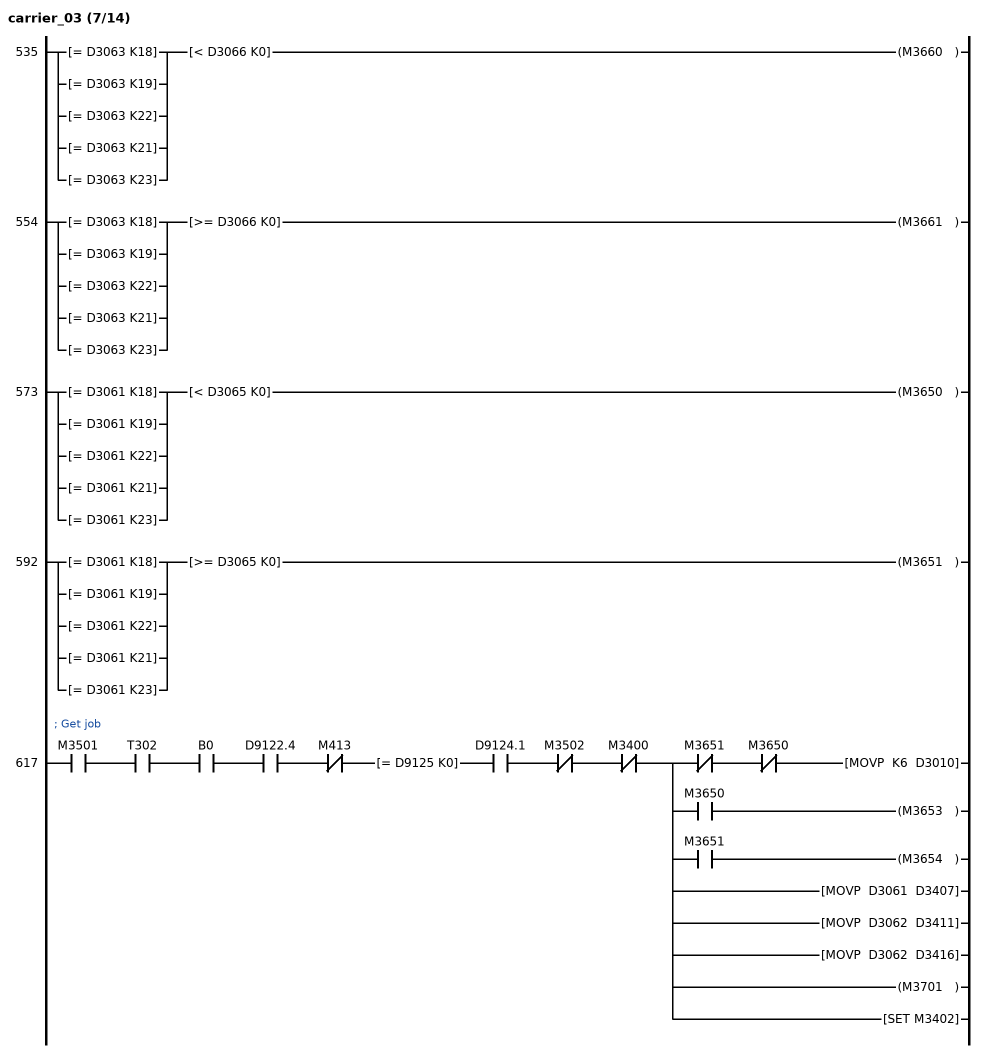
[picture p72: ladder of carrier_03, rungs at steps 535 to 617]
535   LD=     D3063 K18
      OR=     D3063 K19
      OR=     D3063 K22
      OR=     D3063 K21
      OR=     D3063 K23
      AND<    D3066 K0
      OUT     M3660
554   LD=     D3063 K18
      OR=     D3063 K19
      OR=     D3063 K22
      OR=     D3063 K21
      OR=     D3063 K23
      AND>=   D3066 K0
      OUT     M3661
573   LD=     D3061 K18
      OR=     D3061 K19
      OR=     D3061 K22
      OR=     D3061 K21
      OR=     D3061 K23
      AND<    D3065 K0
      OUT     M3650
592   LD=     D3061 K18
      OR=     D3061 K19
      OR=     D3061 K22
      OR=     D3061 K21
      OR=     D3061 K23
      AND>=   D3065 K0
      OUT     M3651
; Get job
617   LD      M3501
      AND     T302
      AND     B0
      AND     D9122.4
      ANI     M413
      AND=    D9125 K0
      AND     D9124.1
      ANI     M3502
      ANI     M3400
      MPS
      ANI     M3651
      ANI     M3650
      MOVP    K6 D3010
      MRD
      AND     M3650
      OUT     M3653
      MRD
      AND     M3651
      OUT     M3654
      MPP
      MOVP    D3061 D3407
      MOVP    D3062 D3411
      MOVP    D3062 D3416
      OUT     M3701
      SET     M3402
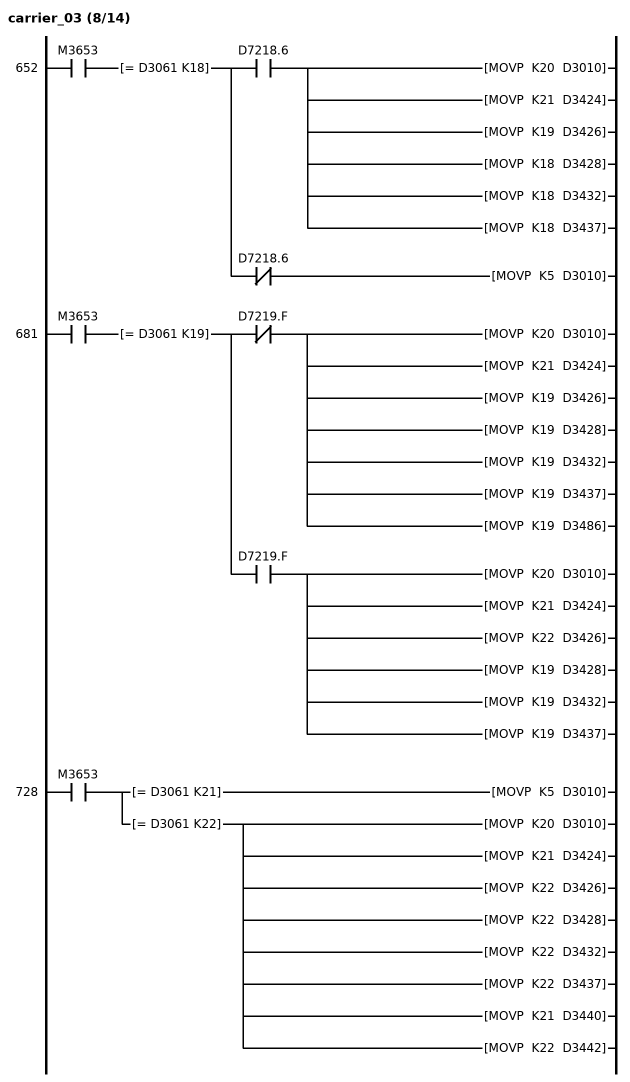
652   LD      M3653
      AND=    D3061 K18
      MPS
      AND     D7218.6
      MOVP    K20 D3010
      MOVP    K21 D3424
      MOVP    K19 D3426
      MOVP    K18 D3428
      MOVP    K18 D3432
      MOVP    K18 D3437
      MPP
      ANI     D7218.6
      MOVP    K5 D3010
681   LD      M3653
      AND=    D3061 K19
      MPS
      ANI     D7219.F
      MOVP    K20 D3010
      MOVP    K21 D3424
      MOVP    K19 D3426
      MOVP    K19 D3428
      MOVP    K19 D3432
      MOVP    K19 D3437
      MOVP    K19 D3486
      MPP
      AND     D7219.F
      MOVP    K20 D3010
      MOVP    K21 D3424
      MOVP    K22 D3426
      MOVP    K19 D3428
      MOVP    K19 D3432
      MOVP    K19 D3437
728   LD      M3653
      MPS
      AND=    D3061 K21
      MOVP    K5 D3010
      MPP
      AND=    D3061 K22
      MOVP    K20 D3010
      MOVP    K21 D3424
      MOVP    K22 D3426
      MOVP    K22 D3428
      MOVP    K22 D3432
      MOVP    K22 D3437
      MOVP    K21 D3440
      MOVP    K22 D3442
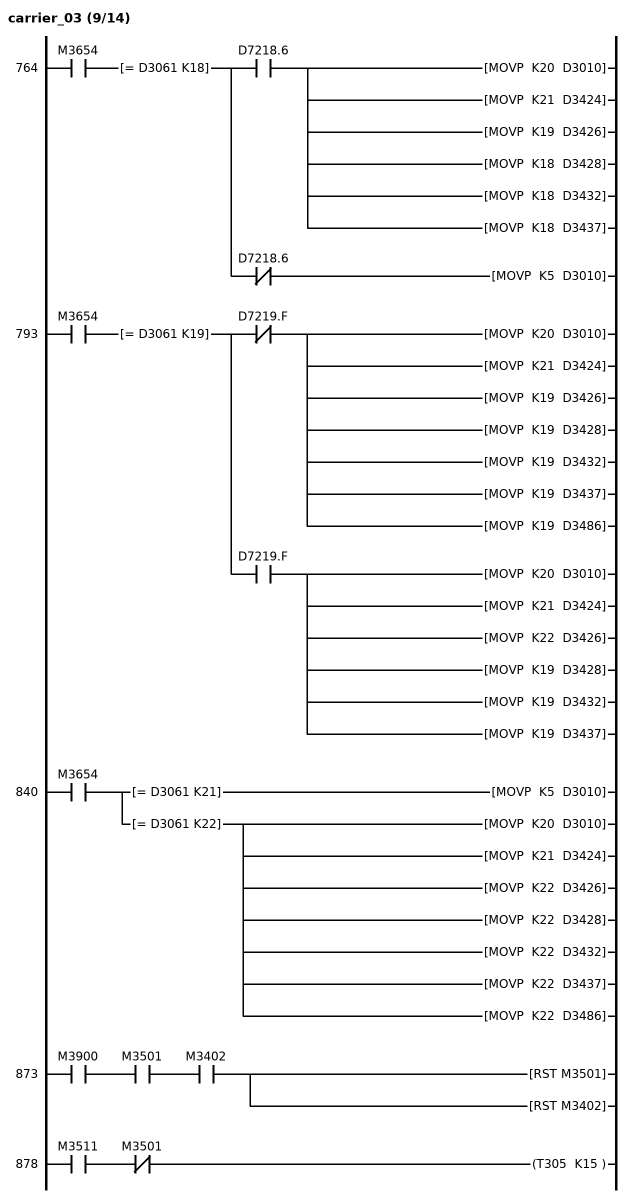
764   LD      M3654
      AND=    D3061 K18
      MPS
      AND     D7218.6
      MOVP    K20 D3010
      MOVP    K21 D3424
      MOVP    K19 D3426
      MOVP    K18 D3428
      MOVP    K18 D3432
      MOVP    K18 D3437
      MPP
      ANI     D7218.6
      MOVP    K5 D3010
793   LD      M3654
      AND=    D3061 K19
      MPS
      ANI     D7219.F
      MOVP    K20 D3010
      MOVP    K21 D3424
      MOVP    K19 D3426
      MOVP    K19 D3428
      MOVP    K19 D3432
      MOVP    K19 D3437
      MOVP    K19 D3486
      MPP
      AND     D7219.F
      MOVP    K20 D3010
      MOVP    K21 D3424
      MOVP    K22 D3426
      MOVP    K19 D3428
      MOVP    K19 D3432
      MOVP    K19 D3437
840   LD      M3654
      MPS
      AND=    D3061 K21
      MOVP    K5 D3010
      MPP
      AND=    D3061 K22
      MOVP    K20 D3010
      MOVP    K21 D3424
      MOVP    K22 D3426
      MOVP    K22 D3428
      MOVP    K22 D3432
      MOVP    K22 D3437
      MOVP    K22 D3486
873   LD      M3900
      AND     M3501
      AND     M3402
      RST     M3501
      RST     M3402
878   LD      M3511
      ANI     M3501
      OUT     T305 K15
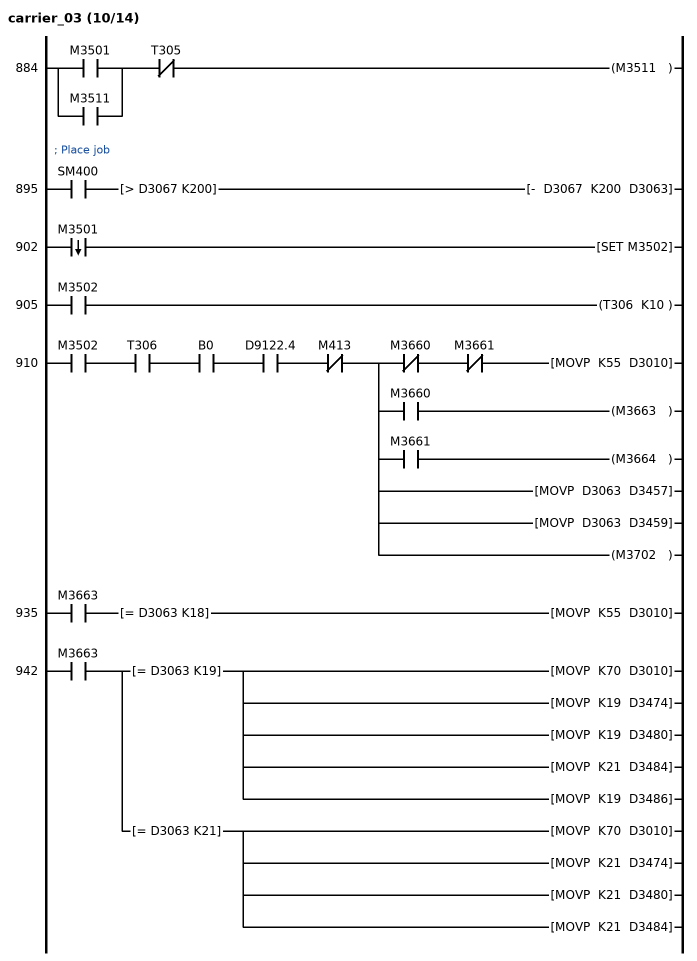
884   LD      M3501
      OR      M3511
      ANI     T305
      OUT     M3511
; Place job
895   LD      SM400
      AND>    D3067 K200
      -       D3067 K200 D3063
902   LDF     M3501
      SET     M3502
905   LD      M3502
      OUT     T306 K10
910   LD      M3502
      AND     T306
      AND     B0
      AND     D9122.4
      ANI     M413
      MPS
      ANI     M3660
      ANI     M3661
      MOVP    K55 D3010
      MRD
      AND     M3660
      OUT     M3663
      MRD
      AND     M3661
      OUT     M3664
      MPP
      MOVP    D3063 D3457
      MOVP    D3063 D3459
      OUT     M3702
935   LD      M3663
      AND=    D3063 K18
      MOVP    K55 D3010
942   LD      M3663
      MPS
      AND=    D3063 K19
      MOVP    K70 D3010
      MOVP    K19 D3474
      MOVP    K19 D3480
      MOVP    K21 D3484
      MOVP    K19 D3486
      MPP
      AND=    D3063 K21
      MOVP    K70 D3010
      MOVP    K21 D3474
      MOVP    K21 D3480
      MOVP    K21 D3484
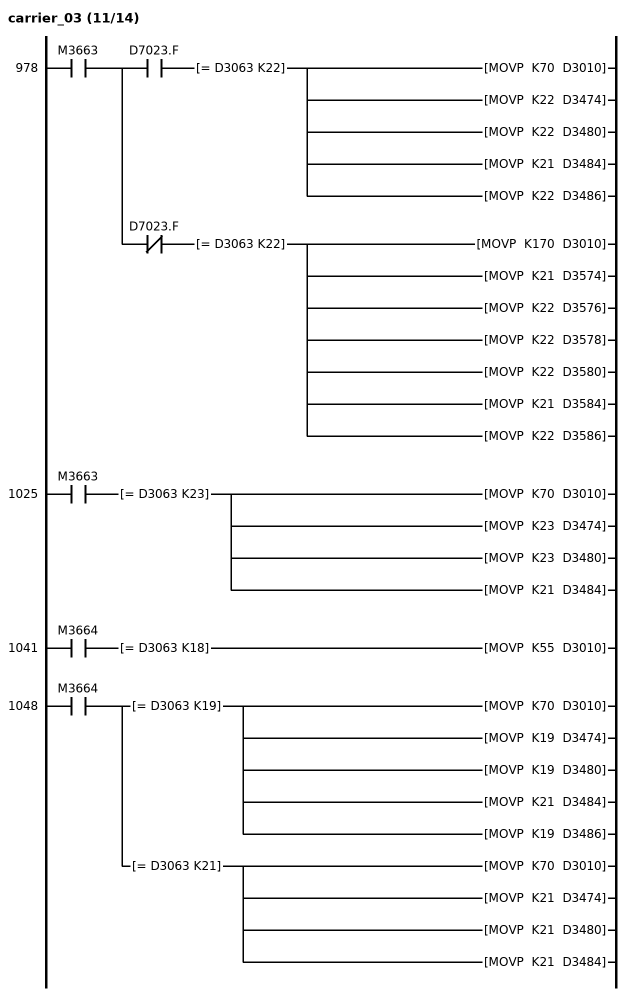
978   LD      M3663
      MPS
      AND     D7023.F
      AND=    D3063 K22
      MOVP    K70 D3010
      MOVP    K22 D3474
      MOVP    K22 D3480
      MOVP    K21 D3484
      MOVP    K22 D3486
      MPP
      ANI     D7023.F
      AND=    D3063 K22
      MOVP    K170 D3010
      MOVP    K21 D3574
      MOVP    K22 D3576
      MOVP    K22 D3578
      MOVP    K22 D3580
      MOVP    K21 D3584
      MOVP    K22 D3586
1025  LD      M3663
      AND=    D3063 K23
      MOVP    K70 D3010
      MOVP    K23 D3474
      MOVP    K23 D3480
      MOVP    K21 D3484
1041  LD      M3664
      AND=    D3063 K18
      MOVP    K55 D3010
1048  LD      M3664
      MPS
      AND=    D3063 K19
      MOVP    K70 D3010
      MOVP    K19 D3474
      MOVP    K19 D3480
      MOVP    K21 D3484
      MOVP    K19 D3486
      MPP
      AND=    D3063 K21
      MOVP    K70 D3010
      MOVP    K21 D3474
      MOVP    K21 D3480
      MOVP    K21 D3484
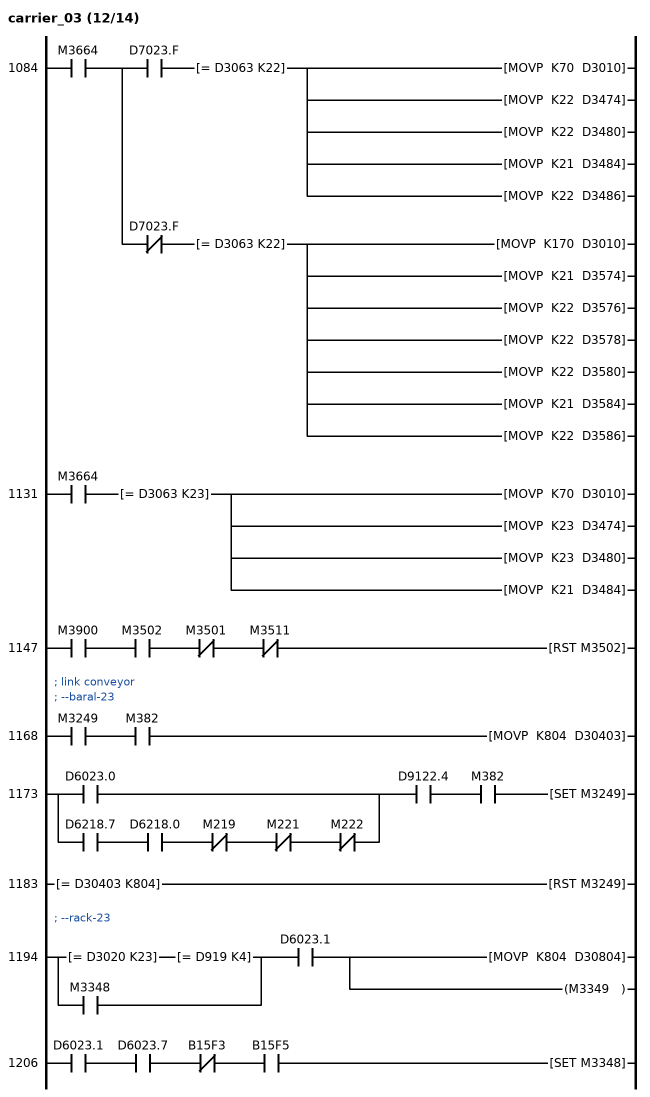
1084  LD      M3664
      MPS
      AND     D7023.F
      AND=    D3063 K22
      MOVP    K70 D3010
      MOVP    K22 D3474
      MOVP    K22 D3480
      MOVP    K21 D3484
      MOVP    K22 D3486
      MPP
      ANI     D7023.F
      AND=    D3063 K22
      MOVP    K170 D3010
      MOVP    K21 D3574
      MOVP    K22 D3576
      MOVP    K22 D3578
      MOVP    K22 D3580
      MOVP    K21 D3584
      MOVP    K22 D3586
1131  LD      M3664
      AND=    D3063 K23
      MOVP    K70 D3010
      MOVP    K23 D3474
      MOVP    K23 D3480
      MOVP    K21 D3484
1147  LD      M3900
      AND     M3502
      ANI     M3501
      ANI     M3511
      RST     M3502
; link conveyor
; --baral-23
1168  LD      M3249
      AND     M382
      MOVP    K804 D30403
1173  LD      D6023.0
      LD      D6218.7
      AND     D6218.0
      ANI     M219
      ANI     M221
      ANI     M222
      ORB
      AND     D9122.4
      AND     M382
      SET     M3249
1183  LD=     D30403 K804
      RST     M3249
; --rack-23
1194  LD=     D3020 K23
      AND=    D919 K4
      OR      M3348
      AND     D6023.1
      MOVP    K804 D30804
      OUT     M3349
1206  LD      D6023.1
      AND     D6023.7
      ANI     B15F3
      AND     B15F5
      SET     M3348
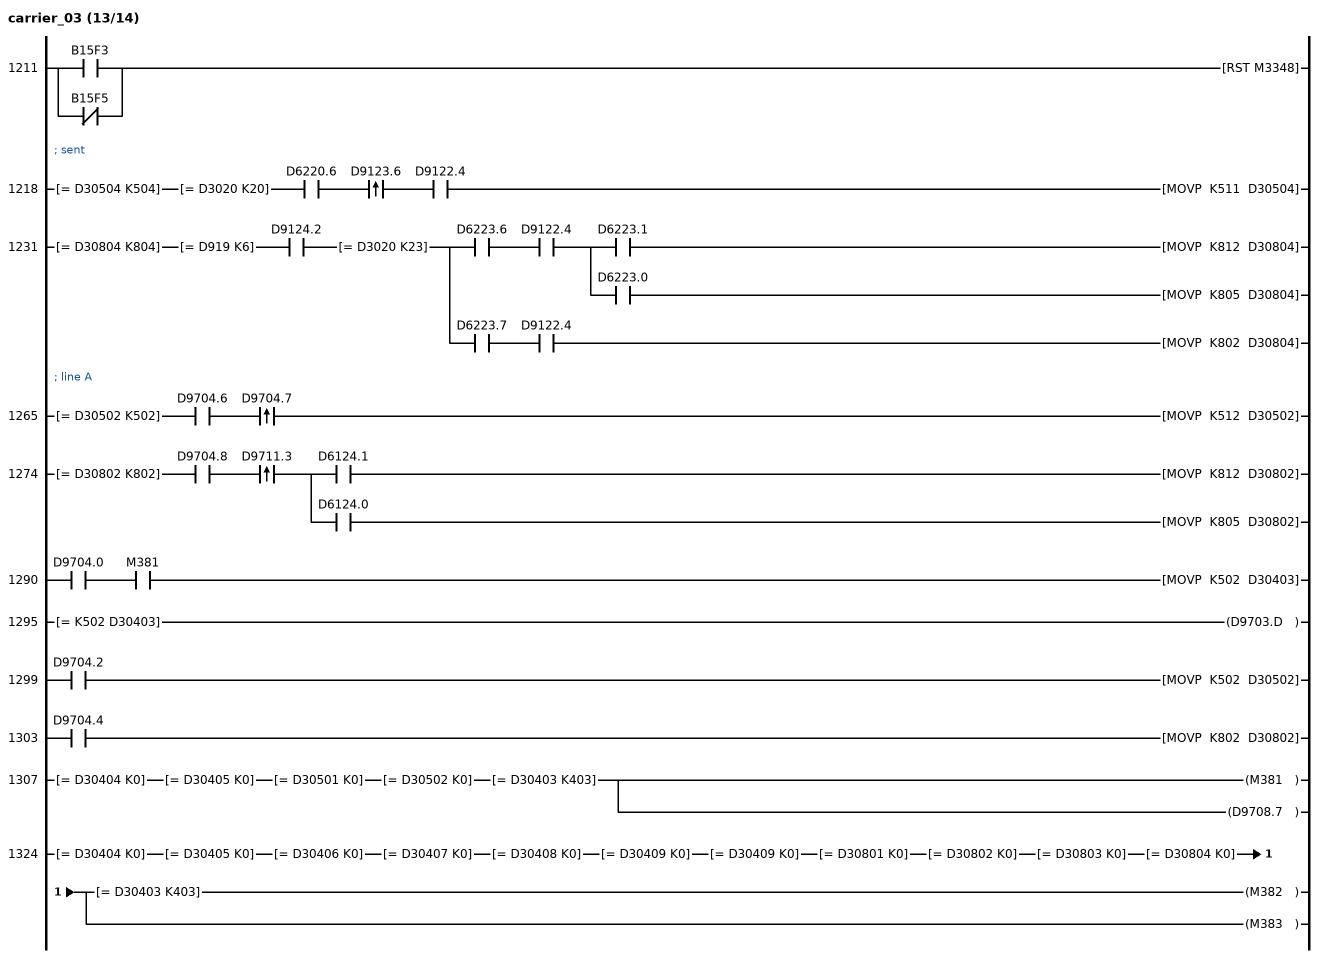
1211  LD      B15F3
      ORI     B15F5
      RST     M3348
; sent
1218  LD=     D30504 K504
      AND=    D3020 K20
      AND     D6220.6
      ANDP    D9123.6
      AND     D9122.4
      MOVP    K511 D30504
1231  LD=     D30804 K804
      AND=    D919 K6
      AND     D9124.2
      AND=    D3020 K23
      MPS
      AND     D6223.6
      AND     D9122.4
      MPS
      AND     D6223.1
      MOVP    K812 D30804
      MPP
      AND     D6223.0
      MOVP    K805 D30804
      MPP
      AND     D6223.7
      AND     D9122.4
      MOVP    K802 D30804
; line A
1265  LD=     D30502 K502
      AND     D9704.6
      ANDP    D9704.7
      MOVP    K512 D30502
1274  LD=     D30802 K802
      AND     D9704.8
      ANDP    D9711.3
      MPS
      AND     D6124.1
      MOVP    K812 D30802
      MPP
      AND     D6124.0
      MOVP    K805 D30802
1290  LD      D9704.0
      AND     M381
      MOVP    K502 D30403
1295  LD=     K502 D30403
      OUT     D9703.D
1299  LD      D9704.2
      MOVP    K502 D30502
1303  LD      D9704.4
      MOVP    K802 D30802
1307  LD=     D30404 K0
      AND=    D30405 K0
      AND=    D30501 K0
      AND=    D30502 K0
      AND=    D30403 K403
      OUT     M381
      OUT     D9708.7
1324  LD=     D30404 K0
      AND=    D30405 K0
      AND=    D30406 K0
      AND=    D30407 K0
      AND=    D30408 K0
      AND=    D30409 K0
      AND=    D30409 K0
      AND=    D30801 K0
      AND=    D30802 K0
      AND=    D30803 K0
      AND=    D30804 K0
      MPS
      AND=    D30403 K403
      OUT     M382
      MPP
      OUT     M383
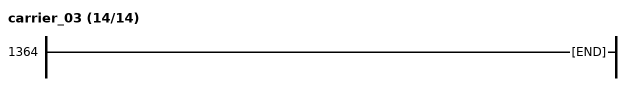
1364  END
END_PROGRAM

PROGRAM carrier_move
0     END
END_PROGRAM

PROGRAM carrier_reset
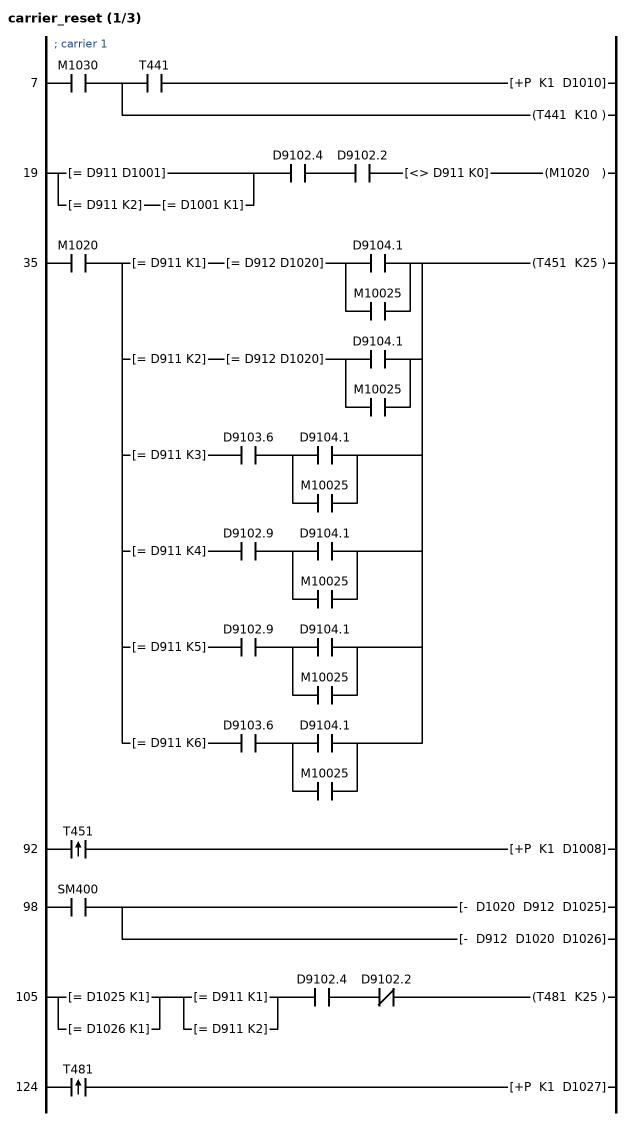
; carrier 1
7     LD      M1030
      MPS
      AND     T441
      +P      K1 D1010
      MPP
      OUT     T441 K10
19    LD=     D911 D1001
      LD=     D911 K2
      AND=    D1001 K1
      ORB
      AND     D9102.4
      AND     D9102.2
      AND<>   D911 K0
      OUT     M1020
35    LD      M1020
      LD=     D911 K1
      AND=    D912 D1020
      LD      D9104.1
      OR      M10025
      ANB
      LD=     D911 K2
      AND=    D912 D1020
      LD      D9104.1
      OR      M10025
      ANB
      ORB
      LD=     D911 K3
      AND     D9103.6
      LD      D9104.1
      OR      M10025
      ANB
      ORB
      LD=     D911 K4
      AND     D9102.9
      LD      D9104.1
      OR      M10025
      ANB
      ORB
      LD=     D911 K5
      AND     D9102.9
      LD      D9104.1
      OR      M10025
      ANB
      ORB
      LD=     D911 K6
      AND     D9103.6
      LD      D9104.1
      OR      M10025
      ANB
      ORB
      ANB
      OUT     T451 K25
92    LDP     T451
      +P      K1 D1008
98    LD      SM400
      -       D1020 D912 D1025
      -       D912 D1020 D1026
105   LD=     D1025 K1
      OR=     D1026 K1
      LD=     D911 K1
      OR=     D911 K2
      ANB
      AND     D9102.4
      ANI     D9102.2
      OUT     T481 K25
124   LDP     T481
      +P      K1 D1027
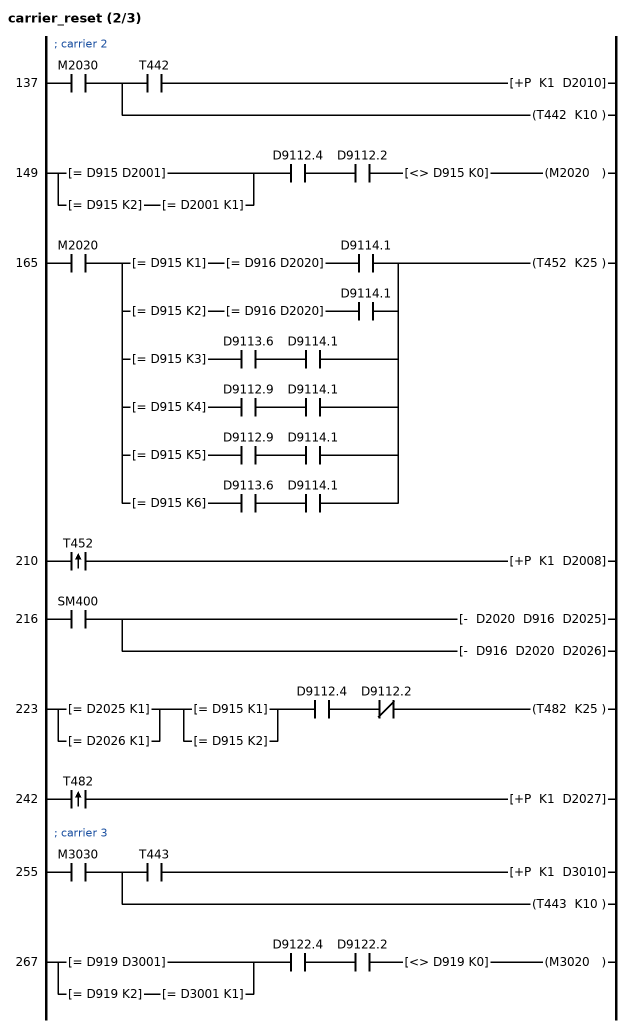
; carrier 2
137   LD      M2030
      MPS
      AND     T442
      +P      K1 D2010
      MPP
      OUT     T442 K10
149   LD=     D915 D2001
      LD=     D915 K2
      AND=    D2001 K1
      ORB
      AND     D9112.4
      AND     D9112.2
      AND<>   D915 K0
      OUT     M2020
165   LD      M2020
      LD=     D915 K1
      AND=    D916 D2020
      AND     D9114.1
      LD=     D915 K2
      AND=    D916 D2020
      AND     D9114.1
      ORB
      LD=     D915 K3
      AND     D9113.6
      AND     D9114.1
      ORB
      LD=     D915 K4
      AND     D9112.9
      AND     D9114.1
      ORB
      LD=     D915 K5
      AND     D9112.9
      AND     D9114.1
      ORB
      LD=     D915 K6
      AND     D9113.6
      AND     D9114.1
      ORB
      ANB
      OUT     T452 K25
210   LDP     T452
      +P      K1 D2008
216   LD      SM400
      -       D2020 D916 D2025
      -       D916 D2020 D2026
223   LD=     D2025 K1
      OR=     D2026 K1
      LD=     D915 K1
      OR=     D915 K2
      ANB
      AND     D9112.4
      ANI     D9112.2
      OUT     T482 K25
242   LDP     T482
      +P      K1 D2027
; carrier 3
255   LD      M3030
      MPS
      AND     T443
      +P      K1 D3010
      MPP
      OUT     T443 K10
267   LD=     D919 D3001
      LD=     D919 K2
      AND=    D3001 K1
      ORB
      AND     D9122.4
      AND     D9122.2
      AND<>   D919 K0
      OUT     M3020
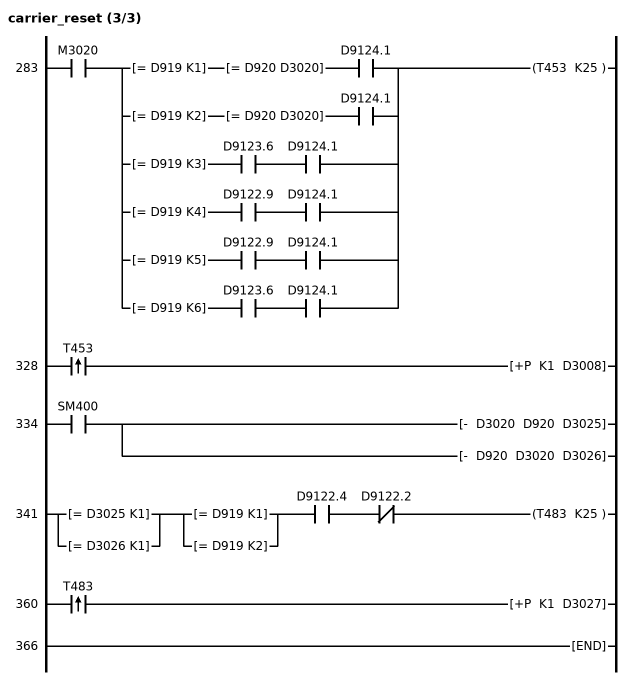
283   LD      M3020
      LD=     D919 K1
      AND=    D920 D3020
      AND     D9124.1
      LD=     D919 K2
      AND=    D920 D3020
      AND     D9124.1
      ORB
      LD=     D919 K3
      AND     D9123.6
      AND     D9124.1
      ORB
      LD=     D919 K4
      AND     D9122.9
      AND     D9124.1
      ORB
      LD=     D919 K5
      AND     D9122.9
      AND     D9124.1
      ORB
      LD=     D919 K6
      AND     D9123.6
      AND     D9124.1
      ORB
      ANB
      OUT     T453 K25
328   LDP     T453
      +P      K1 D3008
334   LD      SM400
      -       D3020 D920 D3025
      -       D920 D3020 D3026
341   LD=     D3025 K1
      OR=     D3026 K1
      LD=     D919 K1
      OR=     D919 K2
      ANB
      AND     D9122.4
      ANI     D9122.2
      OUT     T483 K25
360   LDP     T483
      +P      K1 D3027
366   END
END_PROGRAM

PROGRAM comparater
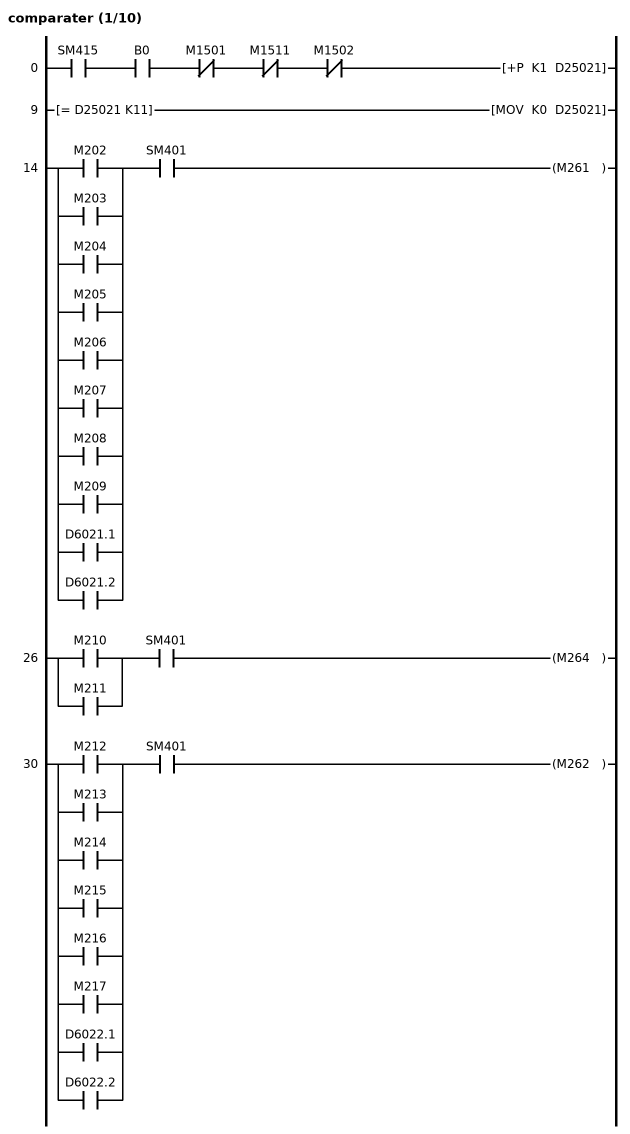
0     LD      SM415
      AND     B0
      ANI     M1501
      ANI     M1511
      ANI     M1502
      +P      K1 D25021
9     LD=     D25021 K11
      MOV     K0 D25021
14    LD      M202
      OR      M203
      OR      M204
      OR      M205
      OR      M206
      OR      M207
      OR      M208
      OR      M209
      OR      D6021.1
      OR      D6021.2
      AND     SM401
      OUT     M261
26    LD      M210
      OR      M211
      AND     SM401
      OUT     M264
30    LD      M212
      OR      M213
      OR      M214
      OR      M215
      OR      M216
      OR      M217
      OR      D6022.1
      OR      D6022.2
      AND     SM401
      OUT     M262
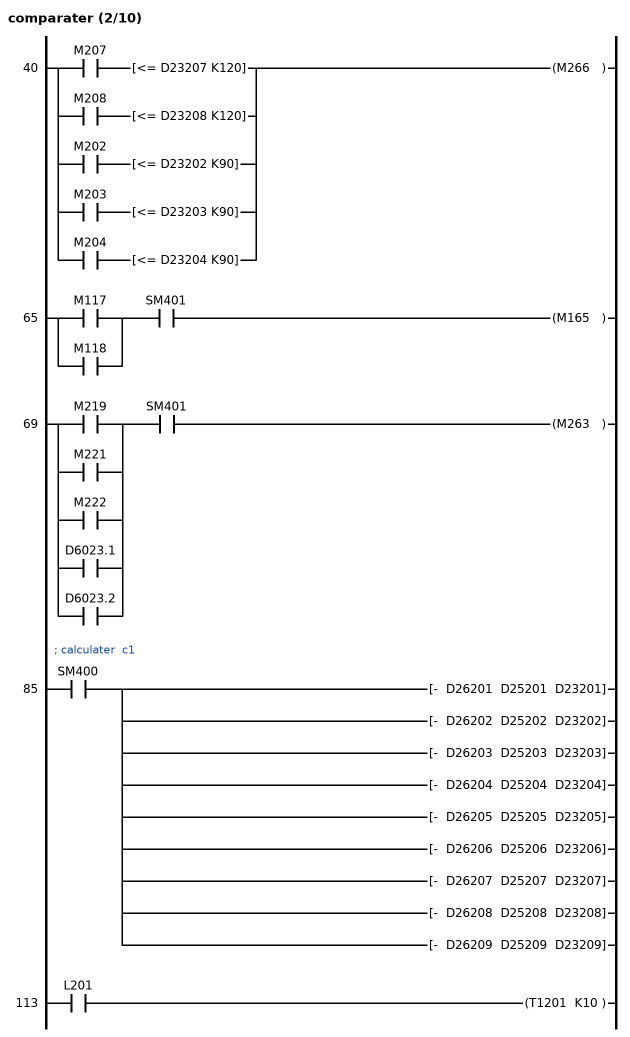
40    LD      M207
      AND<=   D23207 K120
      LD      M208
      AND<=   D23208 K120
      ORB
      LD      M202
      AND<=   D23202 K90
      ORB
      LD      M203
      AND<=   D23203 K90
      ORB
      LD      M204
      AND<=   D23204 K90
      ORB
      OUT     M266
65    LD      M117
      OR      M118
      AND     SM401
      OUT     M165
69    LD      M219
      OR      M221
      OR      M222
      OR      D6023.1
      OR      D6023.2
      AND     SM401
      OUT     M263
; calculater  c1
85    LD      SM400
      -       D26201 D25201 D23201
      -       D26202 D25202 D23202
      -       D26203 D25203 D23203
      -       D26204 D25204 D23204
      -       D26205 D25205 D23205
      -       D26206 D25206 D23206
      -       D26207 D25207 D23207
      -       D26208 D25208 D23208
      -       D26209 D25209 D23209
113   LD      L201
      OUT     T1201 K10
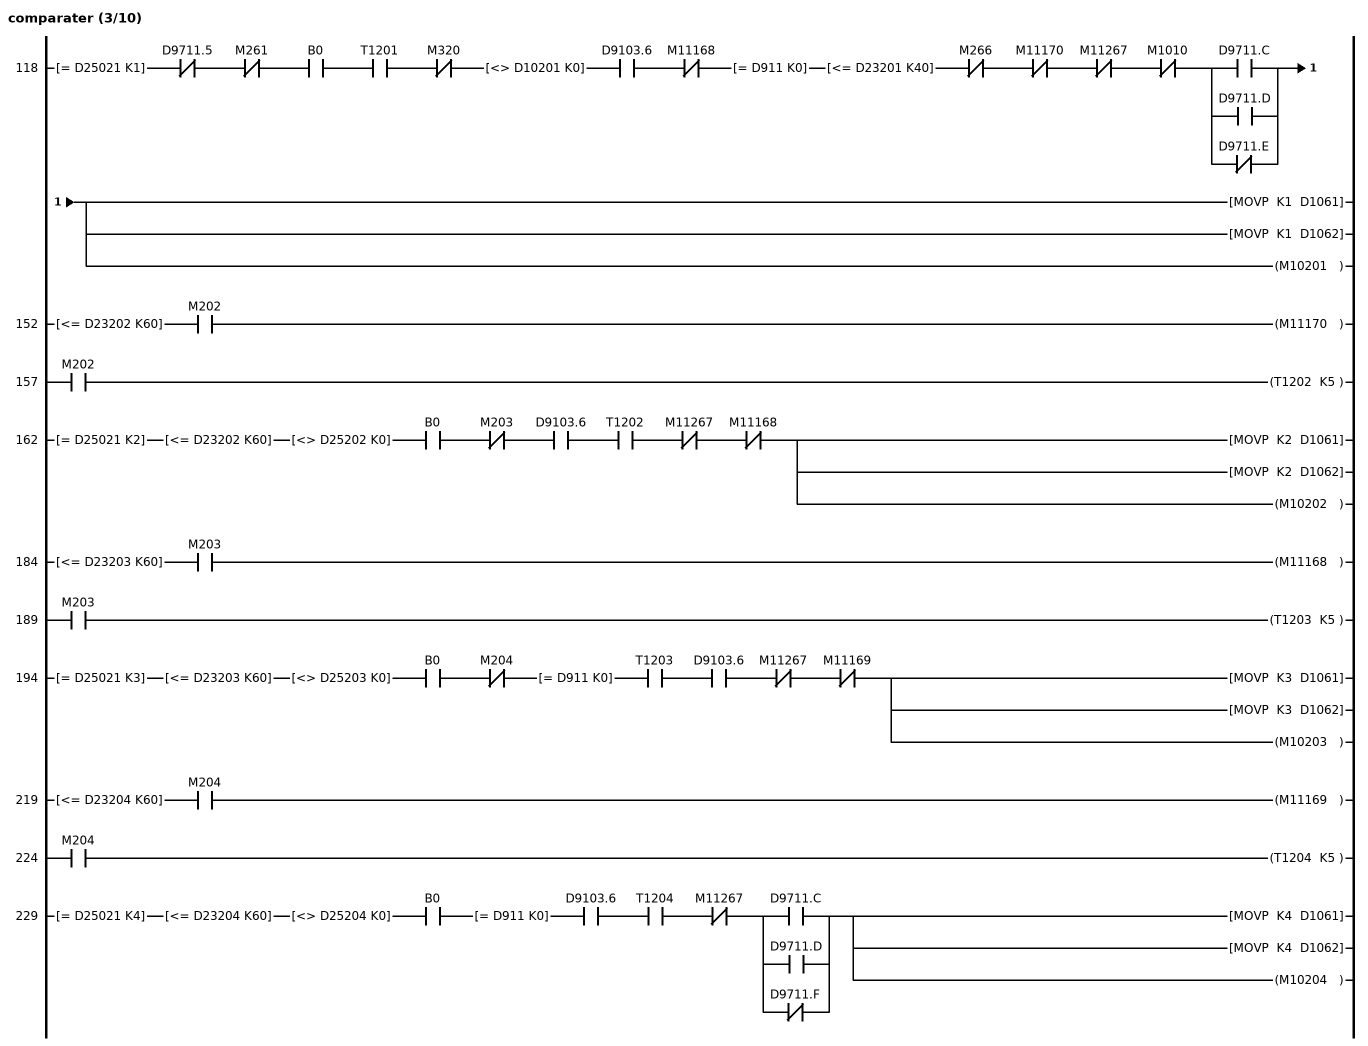
118   LD=     D25021 K1
      ANI     D9711.5
      ANI     M261
      AND     B0
      AND     T1201
      ANI     M320
      AND<>   D10201 K0
      AND     D9103.6
      ANI     M11168
      AND=    D911 K0
      AND<=   D23201 K40
      ANI     M266
      ANI     M11170
      ANI     M11267
      ANI     M1010
      LD      D9711.C
      OR      D9711.D
      ORI     D9711.E
      ANB
      MOVP    K1 D1061
      MOVP    K1 D1062
      OUT     M10201
152   LD<=    D23202 K60
      AND     M202
      OUT     M11170
157   LD      M202
      OUT     T1202 K5
162   LD=     D25021 K2
      AND<=   D23202 K60
      AND<>   D25202 K0
      AND     B0
      ANI     M203
      AND     D9103.6
      AND     T1202
      ANI     M11267
      ANI     M11168
      MOVP    K2 D1061
      MOVP    K2 D1062
      OUT     M10202
184   LD<=    D23203 K60
      AND     M203
      OUT     M11168
189   LD      M203
      OUT     T1203 K5
194   LD=     D25021 K3
      AND<=   D23203 K60
      AND<>   D25203 K0
      AND     B0
      ANI     M204
      AND=    D911 K0
      AND     T1203
      AND     D9103.6
      ANI     M11267
      ANI     M11169
      MOVP    K3 D1061
      MOVP    K3 D1062
      OUT     M10203
219   LD<=    D23204 K60
      AND     M204
      OUT     M11169
224   LD      M204
      OUT     T1204 K5
229   LD=     D25021 K4
      AND<=   D23204 K60
      AND<>   D25204 K0
      AND     B0
      AND=    D911 K0
      AND     D9103.6
      AND     T1204
      ANI     M11267
      LD      D9711.C
      OR      D9711.D
      ORI     D9711.F
      ANB
      MOVP    K4 D1061
      MOVP    K4 D1062
      OUT     M10204
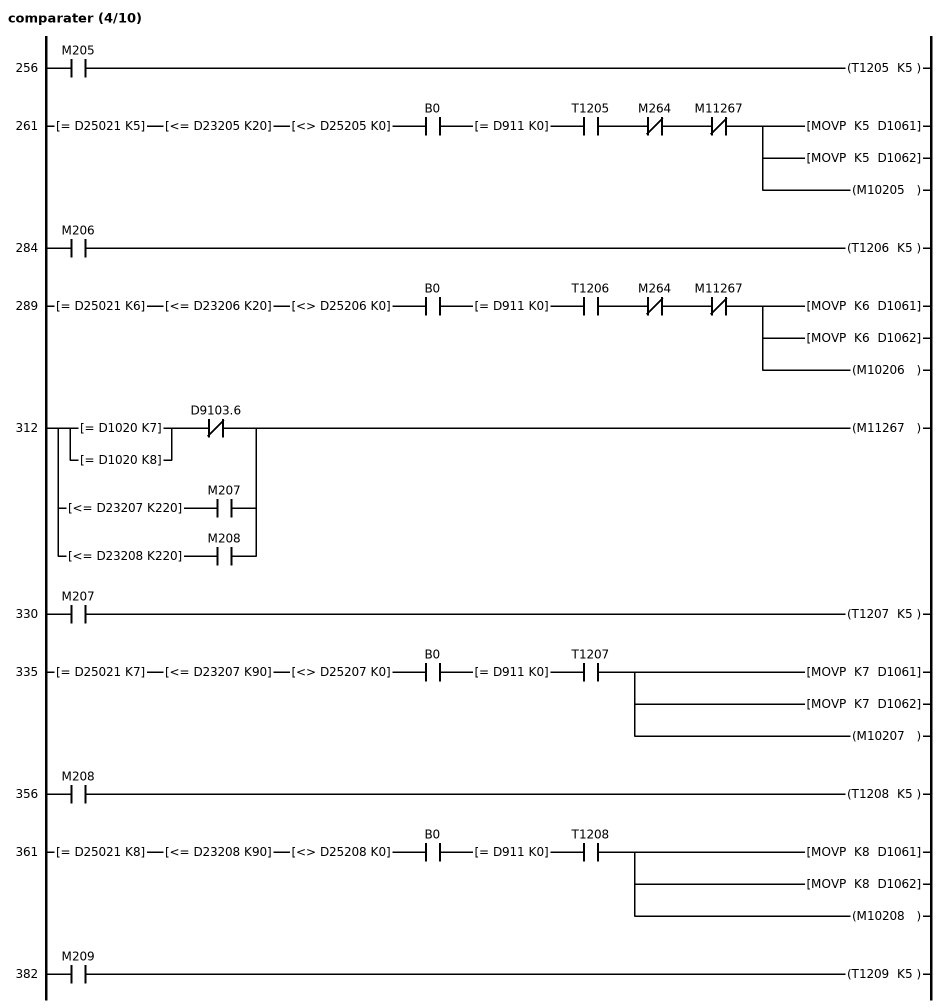
256   LD      M205
      OUT     T1205 K5
261   LD=     D25021 K5
      AND<=   D23205 K20
      AND<>   D25205 K0
      AND     B0
      AND=    D911 K0
      AND     T1205
      ANI     M264
      ANI     M11267
      MOVP    K5 D1061
      MOVP    K5 D1062
      OUT     M10205
284   LD      M206
      OUT     T1206 K5
289   LD=     D25021 K6
      AND<=   D23206 K20
      AND<>   D25206 K0
      AND     B0
      AND=    D911 K0
      AND     T1206
      ANI     M264
      ANI     M11267
      MOVP    K6 D1061
      MOVP    K6 D1062
      OUT     M10206
312   LD=     D1020 K7
      OR=     D1020 K8
      ANI     D9103.6
      LD<=    D23207 K220
      AND     M207
      ORB
      LD<=    D23208 K220
      AND     M208
      ORB
      OUT     M11267
330   LD      M207
      OUT     T1207 K5
335   LD=     D25021 K7
      AND<=   D23207 K90
      AND<>   D25207 K0
      AND     B0
      AND=    D911 K0
      AND     T1207
      MOVP    K7 D1061
      MOVP    K7 D1062
      OUT     M10207
356   LD      M208
      OUT     T1208 K5
361   LD=     D25021 K8
      AND<=   D23208 K90
      AND<>   D25208 K0
      AND     B0
      AND=    D911 K0
      AND     T1208
      MOVP    K8 D1061
      MOVP    K8 D1062
      OUT     M10208
382   LD      M209
      OUT     T1209 K5
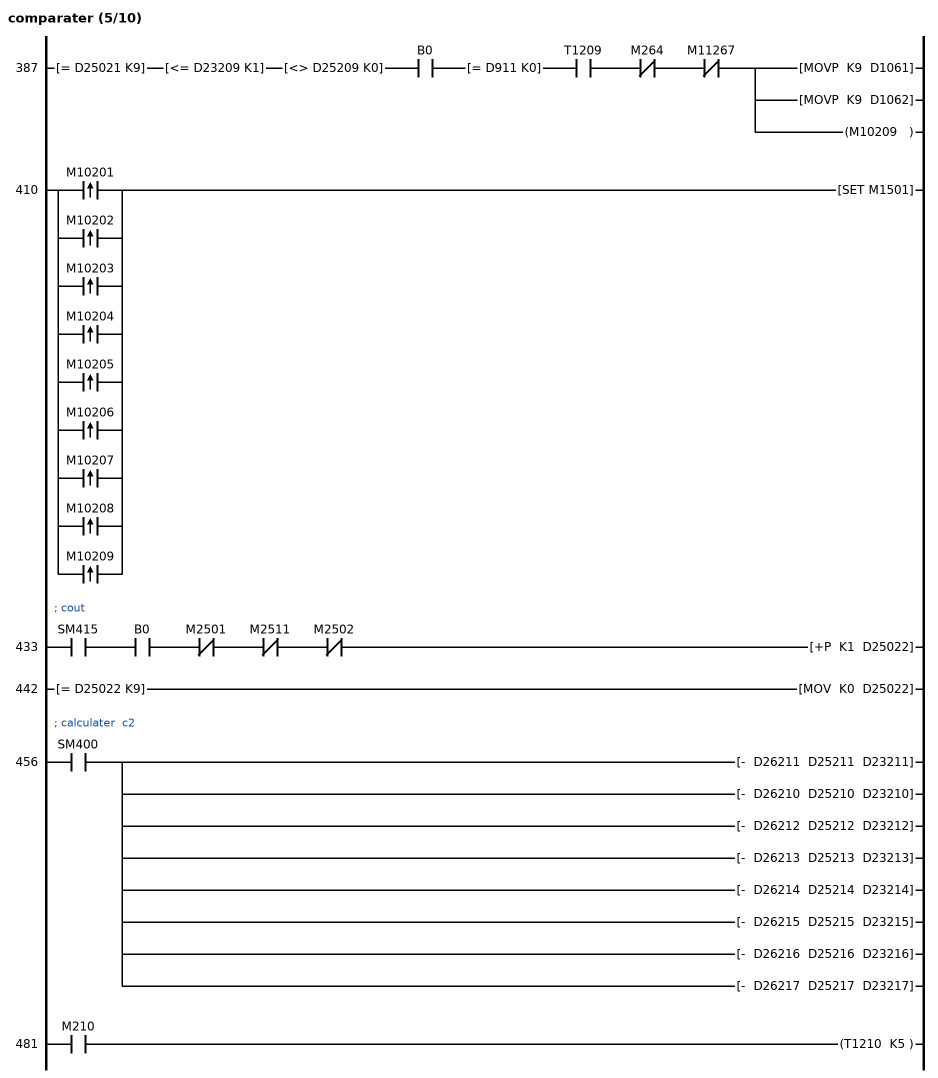
387   LD=     D25021 K9
      AND<=   D23209 K1
      AND<>   D25209 K0
      AND     B0
      AND=    D911 K0
      AND     T1209
      ANI     M264
      ANI     M11267
      MOVP    K9 D1061
      MOVP    K9 D1062
      OUT     M10209
410   LDP     M10201
      ORP     M10202
      ORP     M10203
      ORP     M10204
      ORP     M10205
      ORP     M10206
      ORP     M10207
      ORP     M10208
      ORP     M10209
      SET     M1501
; cout
433   LD      SM415
      AND     B0
      ANI     M2501
      ANI     M2511
      ANI     M2502
      +P      K1 D25022
442   LD=     D25022 K9
      MOV     K0 D25022
; calculater  c2
456   LD      SM400
      -       D26211 D25211 D23211
      -       D26210 D25210 D23210
      -       D26212 D25212 D23212
      -       D26213 D25213 D23213
      -       D26214 D25214 D23214
      -       D26215 D25215 D23215
      -       D26216 D25216 D23216
      -       D26217 D25217 D23217
481   LD      M210
      OUT     T1210 K5
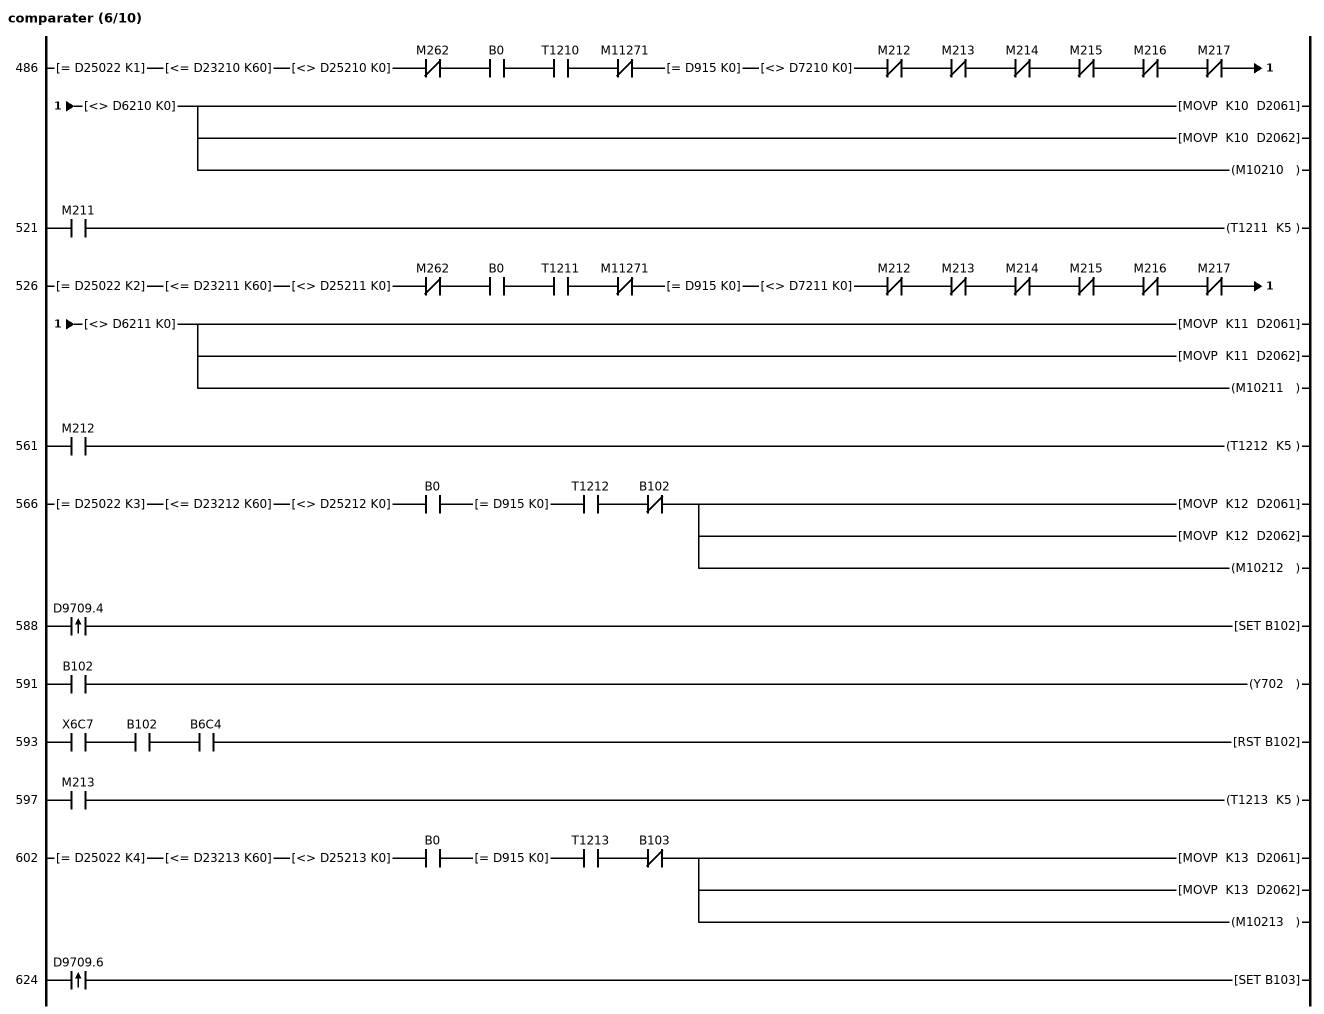
486   LD=     D25022 K1
      AND<=   D23210 K60
      AND<>   D25210 K0
      ANI     M262
      AND     B0
      AND     T1210
      ANI     M11271
      AND=    D915 K0
      AND<>   D7210 K0
      ANI     M212
      ANI     M213
      ANI     M214
      ANI     M215
      ANI     M216
      ANI     M217
      AND<>   D6210 K0
      MOVP    K10 D2061
      MOVP    K10 D2062
      OUT     M10210
521   LD      M211
      OUT     T1211 K5
526   LD=     D25022 K2
      AND<=   D23211 K60
      AND<>   D25211 K0
      ANI     M262
      AND     B0
      AND     T1211
      ANI     M11271
      AND=    D915 K0
      AND<>   D7211 K0
      ANI     M212
      ANI     M213
      ANI     M214
      ANI     M215
      ANI     M216
      ANI     M217
      AND<>   D6211 K0
      MOVP    K11 D2061
      MOVP    K11 D2062
      OUT     M10211
561   LD      M212
      OUT     T1212 K5
566   LD=     D25022 K3
      AND<=   D23212 K60
      AND<>   D25212 K0
      AND     B0
      AND=    D915 K0
      AND     T1212
      ANI     B102
      MOVP    K12 D2061
      MOVP    K12 D2062
      OUT     M10212
588   LDP     D9709.4
      SET     B102
591   LD      B102
      OUT     Y702
593   LD      X6C7
      AND     B102
      AND     B6C4
      RST     B102
597   LD      M213
      OUT     T1213 K5
602   LD=     D25022 K4
      AND<=   D23213 K60
      AND<>   D25213 K0
      AND     B0
      AND=    D915 K0
      AND     T1213
      ANI     B103
      MOVP    K13 D2061
      MOVP    K13 D2062
      OUT     M10213
624   LDP     D9709.6
      SET     B103
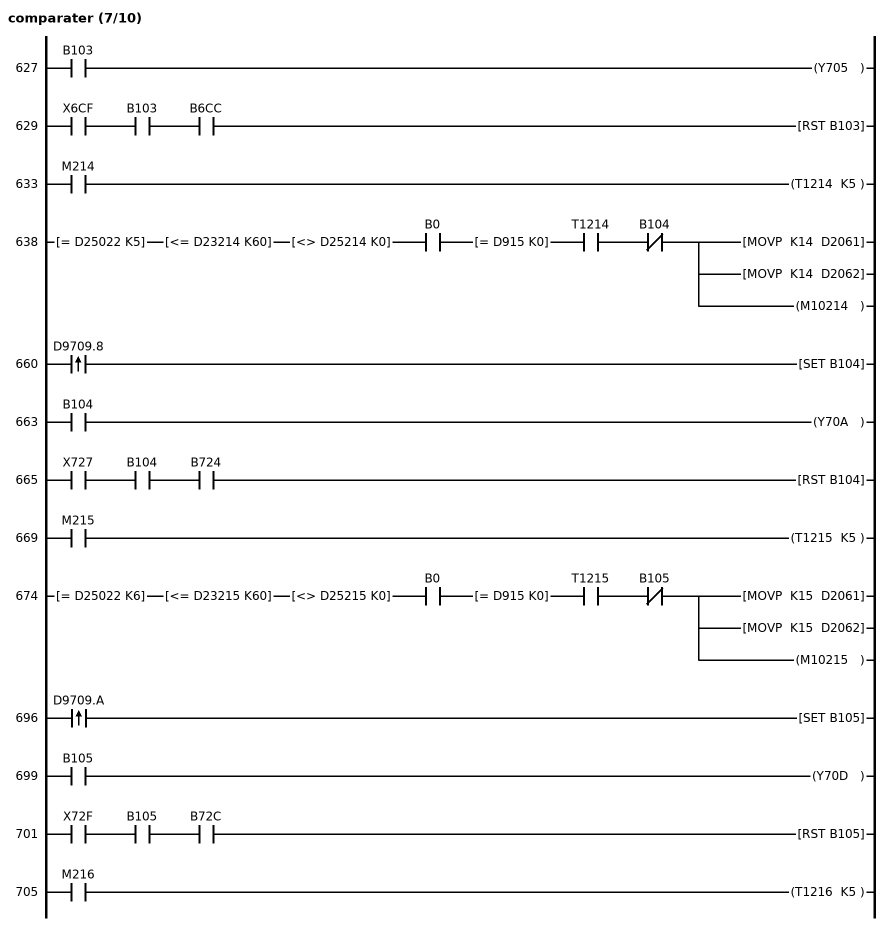
627   LD      B103
      OUT     Y705
629   LD      X6CF
      AND     B103
      AND     B6CC
      RST     B103
633   LD      M214
      OUT     T1214 K5
638   LD=     D25022 K5
      AND<=   D23214 K60
      AND<>   D25214 K0
      AND     B0
      AND=    D915 K0
      AND     T1214
      ANI     B104
      MOVP    K14 D2061
      MOVP    K14 D2062
      OUT     M10214
660   LDP     D9709.8
      SET     B104
663   LD      B104
      OUT     Y70A
665   LD      X727
      AND     B104
      AND     B724
      RST     B104
669   LD      M215
      OUT     T1215 K5
674   LD=     D25022 K6
      AND<=   D23215 K60
      AND<>   D25215 K0
      AND     B0
      AND=    D915 K0
      AND     T1215
      ANI     B105
      MOVP    K15 D2061
      MOVP    K15 D2062
      OUT     M10215
696   LDP     D9709.A
      SET     B105
699   LD      B105
      OUT     Y70D
701   LD      X72F
      AND     B105
      AND     B72C
      RST     B105
705   LD      M216
      OUT     T1216 K5
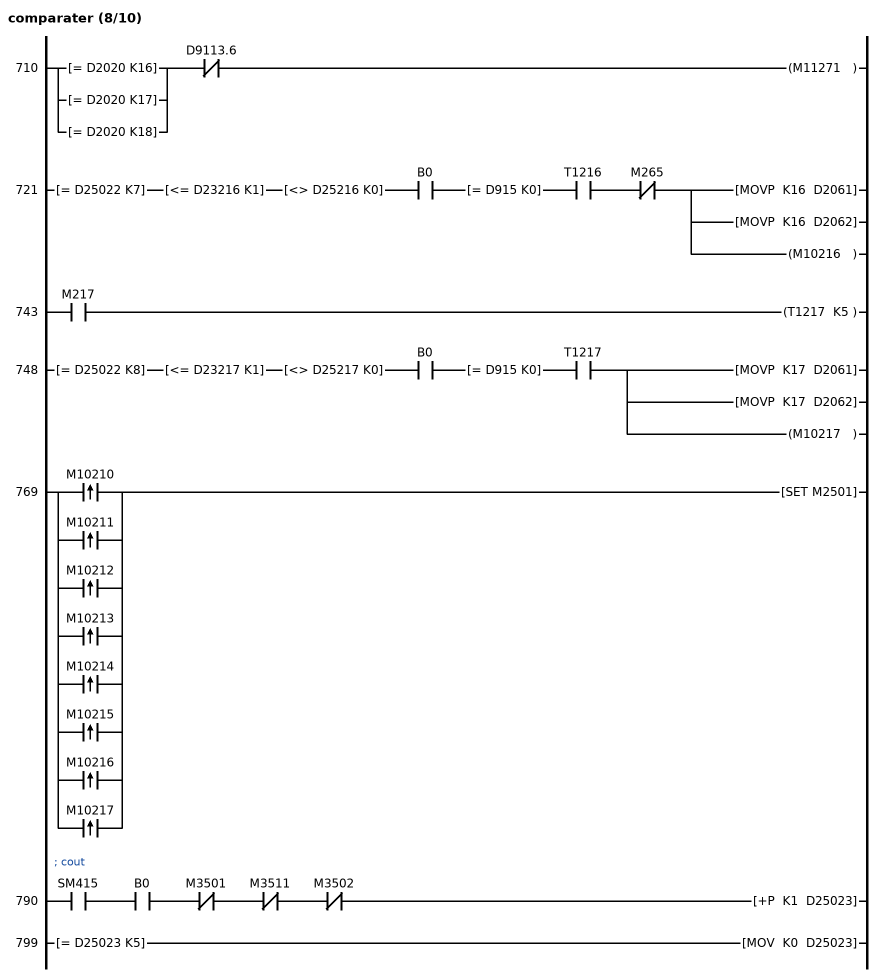
710   LD=     D2020 K16
      OR=     D2020 K17
      OR=     D2020 K18
      ANI     D9113.6
      OUT     M11271
721   LD=     D25022 K7
      AND<=   D23216 K1
      AND<>   D25216 K0
      AND     B0
      AND=    D915 K0
      AND     T1216
      ANI     M265
      MOVP    K16 D2061
      MOVP    K16 D2062
      OUT     M10216
743   LD      M217
      OUT     T1217 K5
748   LD=     D25022 K8
      AND<=   D23217 K1
      AND<>   D25217 K0
      AND     B0
      AND=    D915 K0
      AND     T1217
      MOVP    K17 D2061
      MOVP    K17 D2062
      OUT     M10217
769   LDP     M10210
      ORP     M10211
      ORP     M10212
      ORP     M10213
      ORP     M10214
      ORP     M10215
      ORP     M10216
      ORP     M10217
      SET     M2501
; cout
790   LD      SM415
      AND     B0
      ANI     M3501
      ANI     M3511
      ANI     M3502
      +P      K1 D25023
799   LD=     D25023 K5
      MOV     K0 D25023
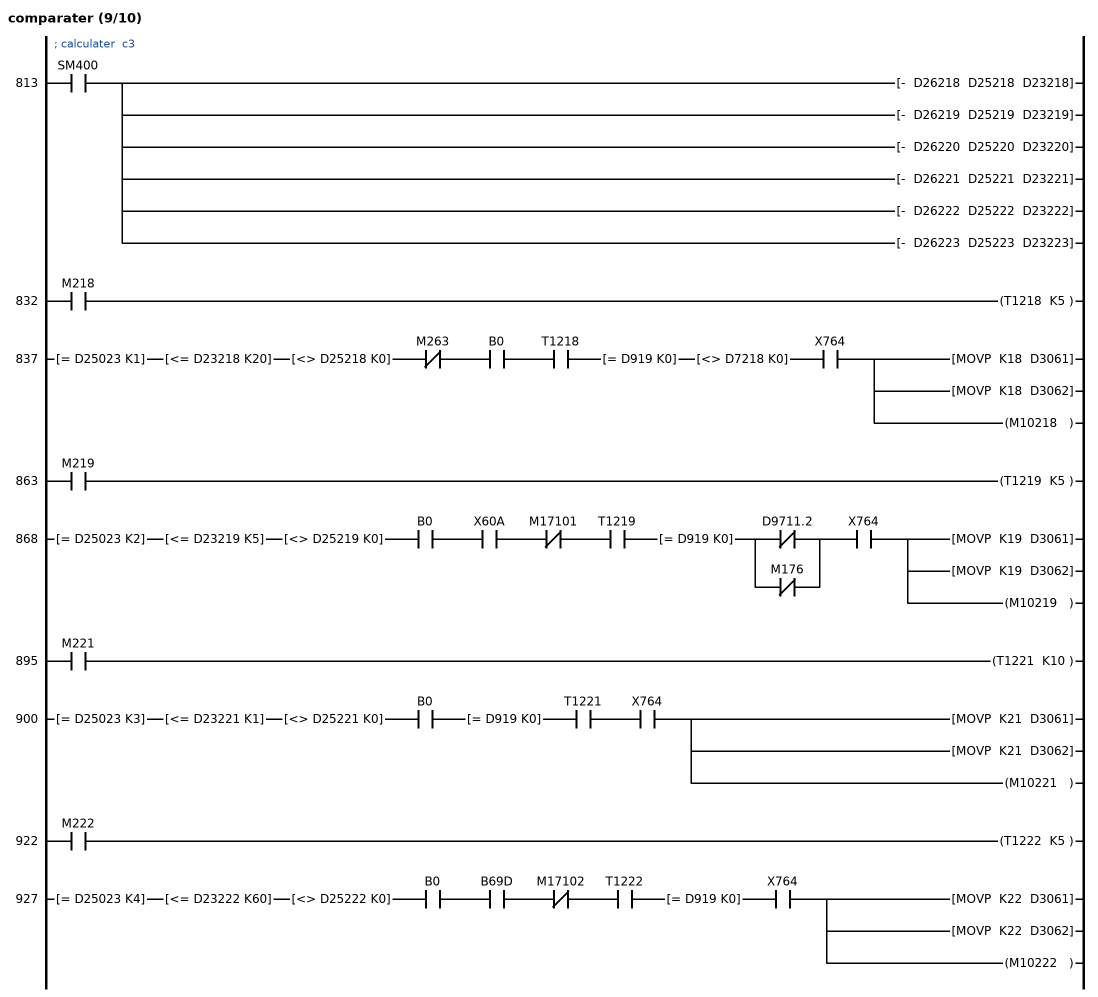
; calculater  c3
813   LD      SM400
      -       D26218 D25218 D23218
      -       D26219 D25219 D23219
      -       D26220 D25220 D23220
      -       D26221 D25221 D23221
      -       D26222 D25222 D23222
      -       D26223 D25223 D23223
832   LD      M218
      OUT     T1218 K5
837   LD=     D25023 K1
      AND<=   D23218 K20
      AND<>   D25218 K0
      ANI     M263
      AND     B0
      AND     T1218
      AND=    D919 K0
      AND<>   D7218 K0
      AND     X764
      MOVP    K18 D3061
      MOVP    K18 D3062
      OUT     M10218
863   LD      M219
      OUT     T1219 K5
868   LD=     D25023 K2
      AND<=   D23219 K5
      AND<>   D25219 K0
      AND     B0
      AND     X60A
      ANI     M17101
      AND     T1219
      AND=    D919 K0
      LDI     D9711.2
      ORI     M176
      ANB
      AND     X764
      MOVP    K19 D3061
      MOVP    K19 D3062
      OUT     M10219
895   LD      M221
      OUT     T1221 K10
900   LD=     D25023 K3
      AND<=   D23221 K1
      AND<>   D25221 K0
      AND     B0
      AND=    D919 K0
      AND     T1221
      AND     X764
      MOVP    K21 D3061
      MOVP    K21 D3062
      OUT     M10221
922   LD      M222
      OUT     T1222 K5
927   LD=     D25023 K4
      AND<=   D23222 K60
      AND<>   D25222 K0
      AND     B0
      AND     B69D
      ANI     M17102
      AND     T1222
      AND=    D919 K0
      AND     X764
      MOVP    K22 D3061
      MOVP    K22 D3062
      OUT     M10222
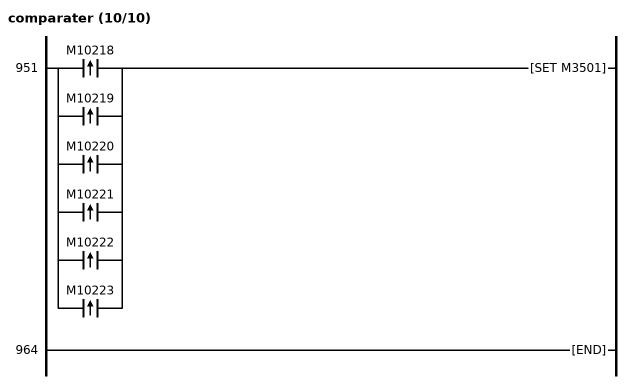
951   LDP     M10218
      ORP     M10219
      ORP     M10220
      ORP     M10221
      ORP     M10222
      ORP     M10223
      SET     M3501
964   END
END_PROGRAM

PROGRAM conveyer_input
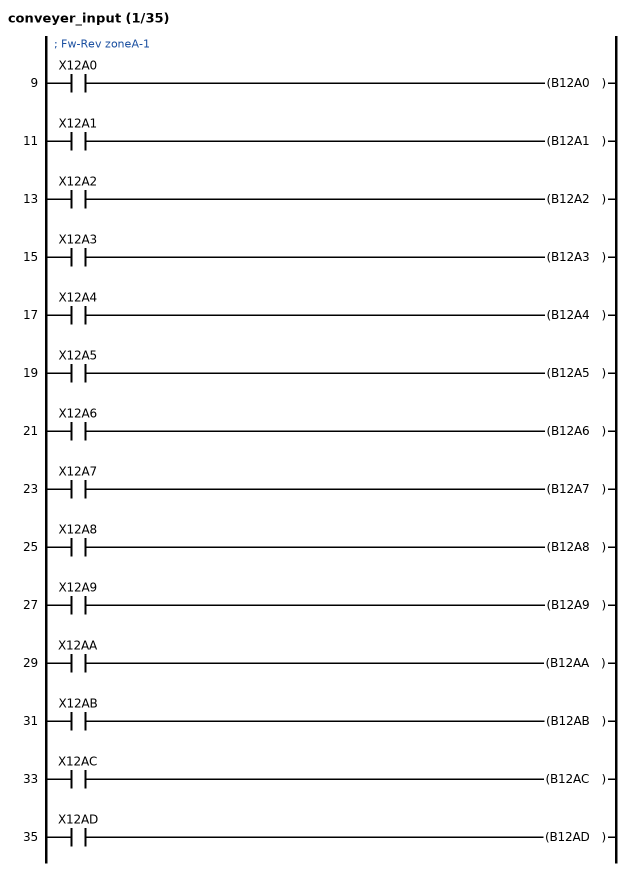
; Fw-Rev zoneA-1
9     LD      X12A0
      OUT     B12A0
11    LD      X12A1
      OUT     B12A1
13    LD      X12A2
      OUT     B12A2
15    LD      X12A3
      OUT     B12A3
17    LD      X12A4
      OUT     B12A4
19    LD      X12A5
      OUT     B12A5
21    LD      X12A6
      OUT     B12A6
23    LD      X12A7
      OUT     B12A7
25    LD      X12A8
      OUT     B12A8
27    LD      X12A9
      OUT     B12A9
29    LD      X12AA
      OUT     B12AA
31    LD      X12AB
      OUT     B12AB
33    LD      X12AC
      OUT     B12AC
35    LD      X12AD
      OUT     B12AD
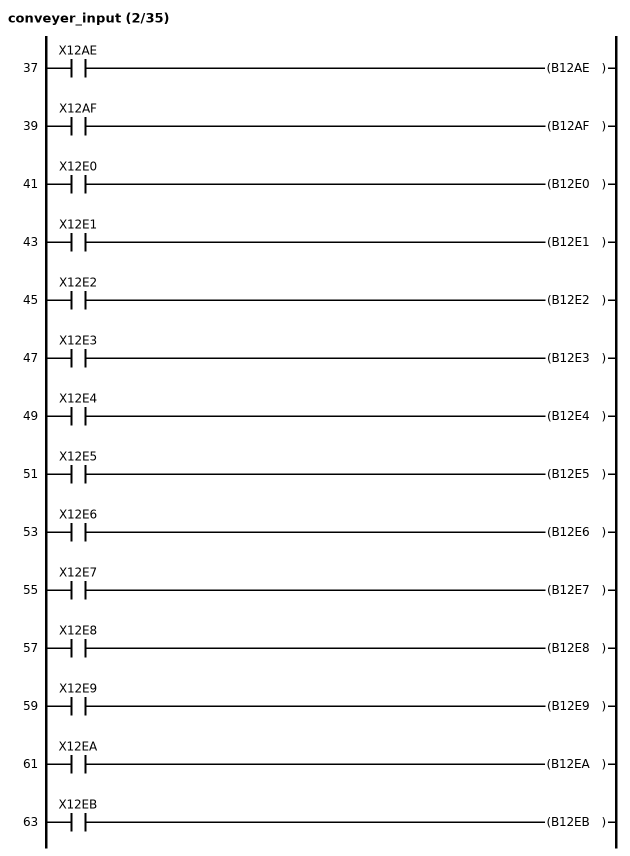
37    LD      X12AE
      OUT     B12AE
39    LD      X12AF
      OUT     B12AF
41    LD      X12E0
      OUT     B12E0
43    LD      X12E1
      OUT     B12E1
45    LD      X12E2
      OUT     B12E2
47    LD      X12E3
      OUT     B12E3
49    LD      X12E4
      OUT     B12E4
51    LD      X12E5
      OUT     B12E5
53    LD      X12E6
      OUT     B12E6
55    LD      X12E7
      OUT     B12E7
57    LD      X12E8
      OUT     B12E8
59    LD      X12E9
      OUT     B12E9
61    LD      X12EA
      OUT     B12EA
63    LD      X12EB
      OUT     B12EB
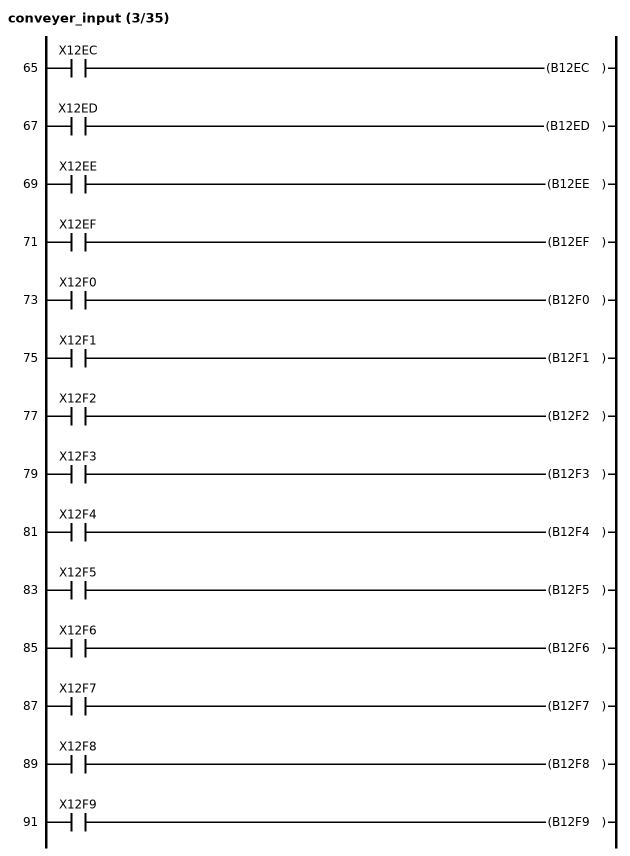
65    LD      X12EC
      OUT     B12EC
67    LD      X12ED
      OUT     B12ED
69    LD      X12EE
      OUT     B12EE
71    LD      X12EF
      OUT     B12EF
73    LD      X12F0
      OUT     B12F0
75    LD      X12F1
      OUT     B12F1
77    LD      X12F2
      OUT     B12F2
79    LD      X12F3
      OUT     B12F3
81    LD      X12F4
      OUT     B12F4
83    LD      X12F5
      OUT     B12F5
85    LD      X12F6
      OUT     B12F6
87    LD      X12F7
      OUT     B12F7
89    LD      X12F8
      OUT     B12F8
91    LD      X12F9
      OUT     B12F9
